// Mitsubishi GX Works2 project: 2023-06-26 #2 생산자동화기능사 14번   PLC: Q03UDV
// 생산자동화기능사

// global labels: Global1
VAR_GLOBAL
  PB1 AT X0 : BOOL;
  PB2 AT X1 : BOOL;
  정지 AT X2 : BOOL;
  공급후진 AT X3 : BOOL;
  공급전진 AT X4 : BOOL;
  가공후진 AT X5 : BOOL;
  가공전진 AT X6 : BOOL;
  송출후진 AT X7 : BOOL;
  송출전진 AT X8 : BOOL;
  배출후진 AT X9 : BOOL;
  배출전진 AT X0A : BOOL;
  매거진 AT X0B : BOOL;
  금속센서 AT X0F : BOOL;
  PB3 AT X10 : BOOL;
  적색 AT Y20 : BOOL;
  황색 AT Y21 : BOOL;
  녹색 AT Y22 : BOOL;
  공급1 AT Y23 : BOOL;
  공급2 AT Y24 : BOOL;
  가공 AT Y25 : BOOL;
  드릴 AT Y26 : BOOL;
  송출 AT Y27 : BOOL;
  배출 AT Y28 : BOOL;
  컨베이어 AT Y29 : BOOL;
END_VAR

PROGRAM 테스트동작
VAR
  PHASE : INT;
END_VAR
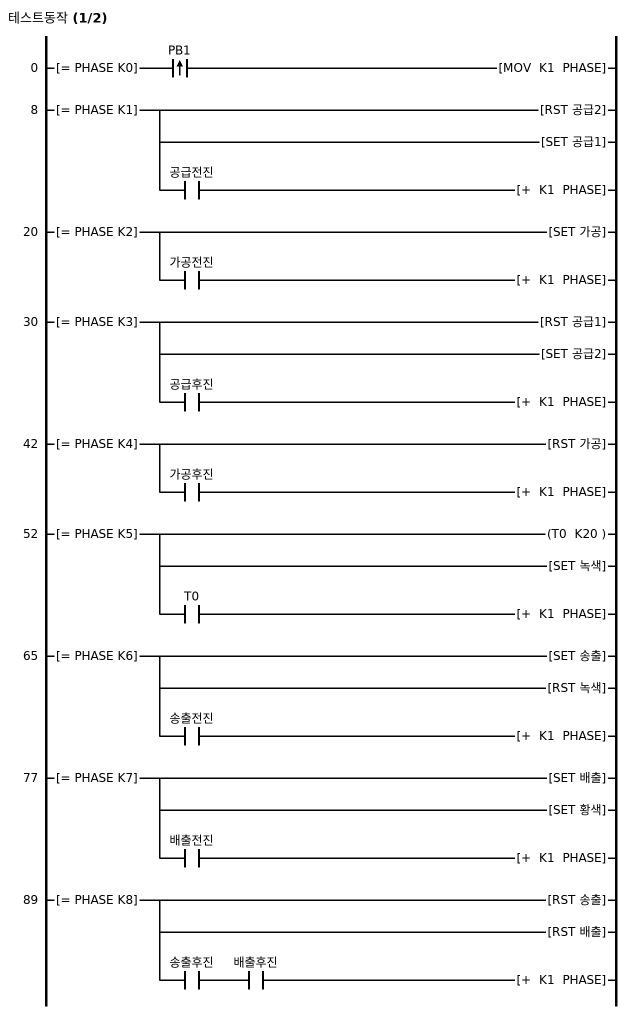
0     LD=     PHASE K0
      ANDP    PB1
      MOV     K1 PHASE
8     LD=     PHASE K1
      RST     공급2
      SET     공급1
      AND     공급전진
      +       K1 PHASE
20    LD=     PHASE K2
      SET     가공
      AND     가공전진
      +       K1 PHASE
30    LD=     PHASE K3
      RST     공급1
      SET     공급2
      AND     공급후진
      +       K1 PHASE
42    LD=     PHASE K4
      RST     가공
      AND     가공후진
      +       K1 PHASE
52    LD=     PHASE K5
      OUT     T0 K20
      SET     녹색
      AND     T0
      +       K1 PHASE
65    LD=     PHASE K6
      SET     송출
      RST     녹색
      AND     송출전진
      +       K1 PHASE
77    LD=     PHASE K7
      SET     배출
      SET     황색
      AND     배출전진
      +       K1 PHASE
89    LD=     PHASE K8
      RST     송출
      RST     배출
      AND     송출후진
      AND     배출후진
      +       K1 PHASE
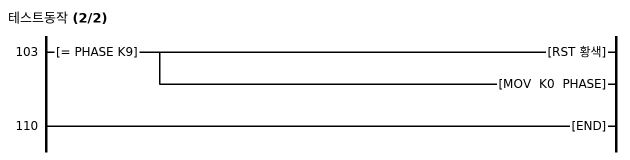
103   LD=     PHASE K9
      RST     황색
      MOV     K0 PHASE
110   END
END_PROGRAM

PROGRAM 단속및연속동작
VAR
  PHASE : INT;
  MODE : INT;
END_VAR
VAR CONSTANT
  단속 : INT;
  연속 : INT := 1;
END_VAR
VAR
  METAL : INT;
END_VAR
VAR CONSTANT
  금속 : INT := 1;
  비금속 : INT := 2;
END_VAR
VAR
  BLINK : ARRAY [0..7] OF BOOL;
  EMG : INT;
END_VAR
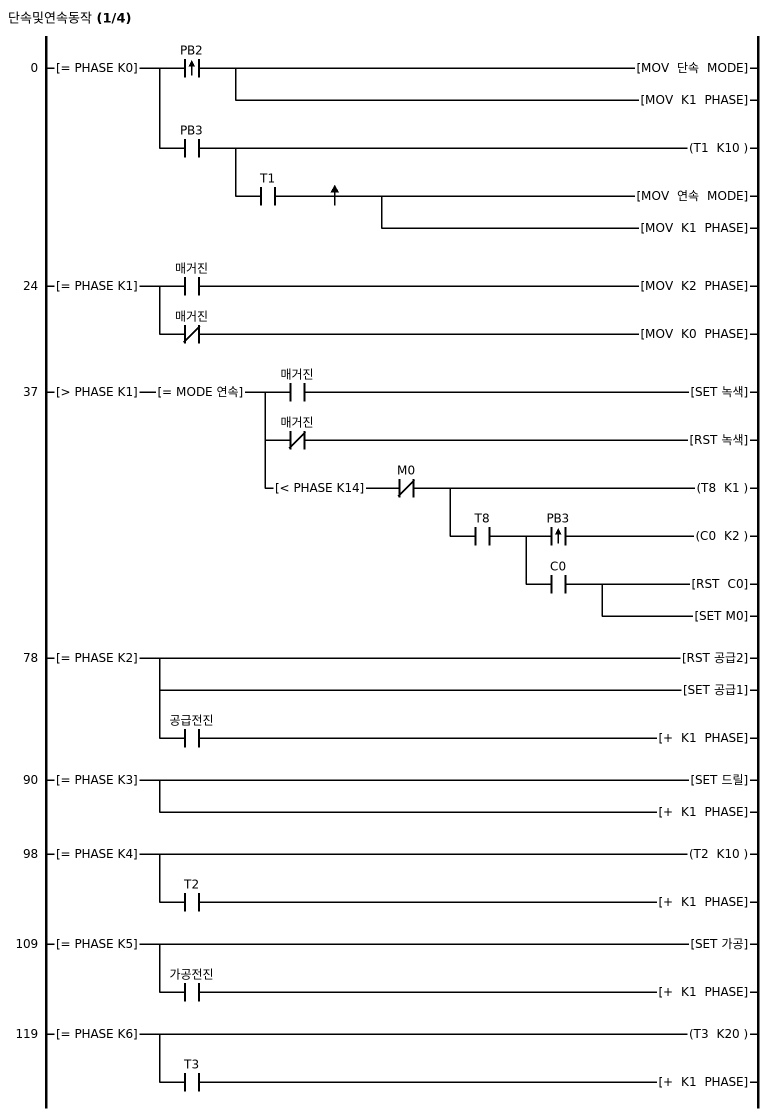
0     LD=     PHASE K0
      MPS
      ANDP    PB2
      MOV     단속 MODE
      MOV     K1 PHASE
      MPP
      AND     PB3
      OUT     T1 K10
      AND     T1
      MEP
      MOV     연속 MODE
      MOV     K1 PHASE
24    LD=     PHASE K1
      MPS
      AND     매거진
      MOV     K2 PHASE
      MPP
      ANI     매거진
      MOV     K0 PHASE
37    LD>     PHASE K1
      AND=    MODE 연속
      MPS
      AND     매거진
      SET     녹색
      MRD
      ANI     매거진
      RST     녹색
      MPP
      AND<    PHASE K14
      ANI     M0
      OUT     T8 K1
      AND     T8
      MPS
      ANDP    PB3
      OUT     C0 K2
      MPP
      AND     C0
      RST     C0
      SET     M0
78    LD=     PHASE K2
      RST     공급2
      SET     공급1
      AND     공급전진
      +       K1 PHASE
90    LD=     PHASE K3
      SET     드릴
      +       K1 PHASE
98    LD=     PHASE K4
      OUT     T2 K10
      AND     T2
      +       K1 PHASE
109   LD=     PHASE K5
      SET     가공
      AND     가공전진
      +       K1 PHASE
119   LD=     PHASE K6
      OUT     T3 K20
      AND     T3
      +       K1 PHASE
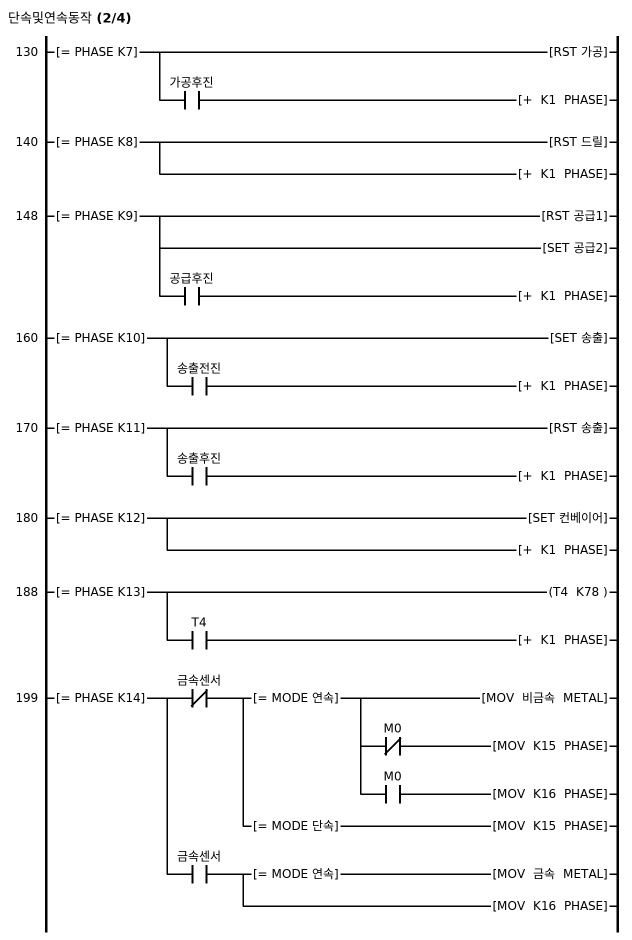
130   LD=     PHASE K7
      RST     가공
      AND     가공후진
      +       K1 PHASE
140   LD=     PHASE K8
      RST     드릴
      +       K1 PHASE
148   LD=     PHASE K9
      RST     공급1
      SET     공급2
      AND     공급후진
      +       K1 PHASE
160   LD=     PHASE K10
      SET     송출
      AND     송출전진
      +       K1 PHASE
170   LD=     PHASE K11
      RST     송출
      AND     송출후진
      +       K1 PHASE
180   LD=     PHASE K12
      SET     컨베이어
      +       K1 PHASE
188   LD=     PHASE K13
      OUT     T4 K78
      AND     T4
      +       K1 PHASE
199   LD=     PHASE K14
      MPS
      ANI     금속센서
      MPS
      AND=    MODE 연속
      MOV     비금속 METAL
      MPS
      ANI     M0
      MOV     K15 PHASE
      MPP
      AND     M0
      MOV     K16 PHASE
      MPP
      AND=    MODE 단속
      MOV     K15 PHASE
      MPP
      AND     금속센서
      MPS
      AND=    MODE 연속
      MOV     금속 METAL
      MPP
      MOV     K16 PHASE
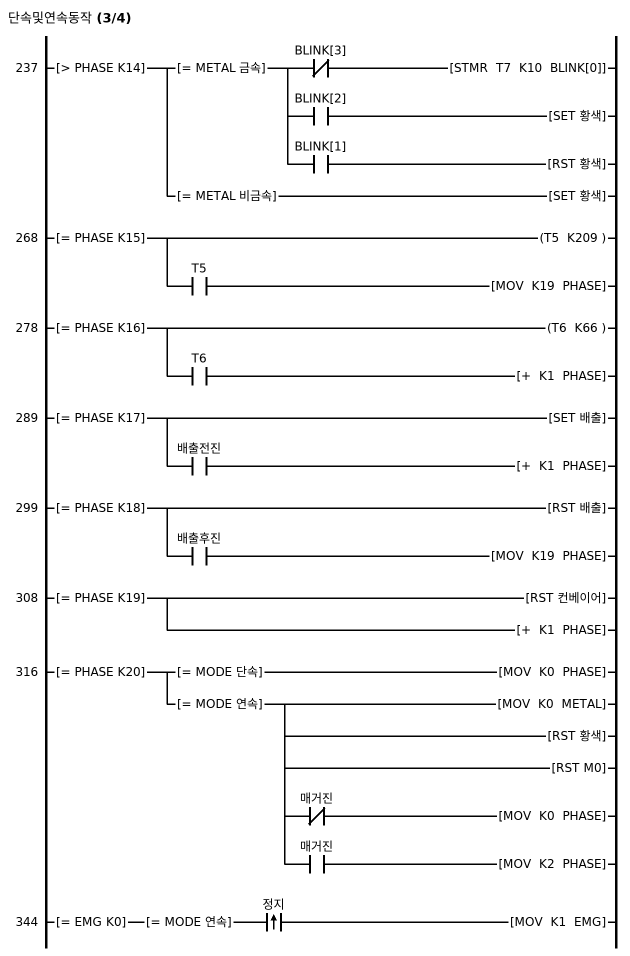
237   LD>     PHASE K14
      MPS
      AND=    METAL 금속
      MPS
      ANI     BLINK[3]
      STMR    T7 K10 BLINK[0]
      MRD
      AND     BLINK[2]
      SET     황색
      MPP
      AND     BLINK[1]
      RST     황색
      MPP
      AND=    METAL 비금속
      SET     황색
268   LD=     PHASE K15
      OUT     T5 K209
      AND     T5
      MOV     K19 PHASE
278   LD=     PHASE K16
      OUT     T6 K66
      AND     T6
      +       K1 PHASE
289   LD=     PHASE K17
      SET     배출
      AND     배출전진
      +       K1 PHASE
299   LD=     PHASE K18
      RST     배출
      AND     배출후진
      MOV     K19 PHASE
308   LD=     PHASE K19
      RST     컨베이어
      +       K1 PHASE
316   LD=     PHASE K20
      MPS
      AND=    MODE 단속
      MOV     K0 PHASE
      MPP
      AND=    MODE 연속
      MOV     K0 METAL
      RST     황색
      RST     M0
      MPS
      ANI     매거진
      MOV     K0 PHASE
      MPP
      AND     매거진
      MOV     K2 PHASE
344   LD=     EMG K0
      AND=    MODE 연속
      ANDP    정지
      MOV     K1 EMG
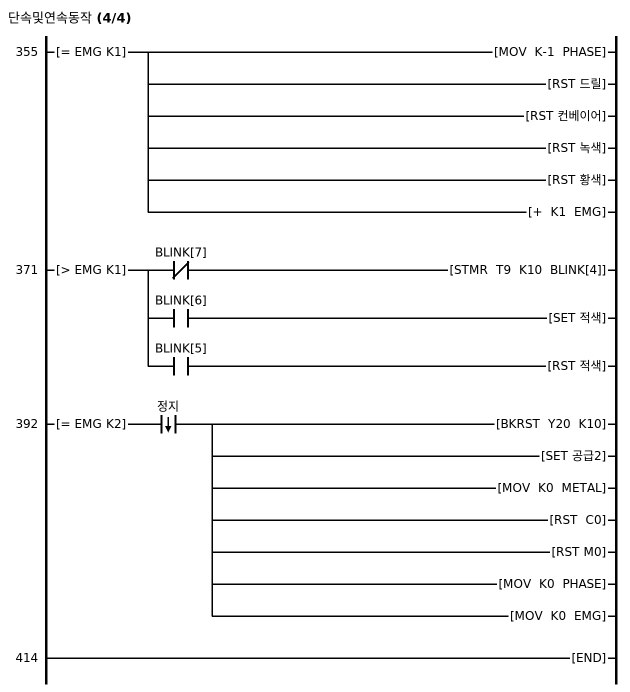
355   LD=     EMG K1
      MOV     K-1 PHASE
      RST     드릴
      RST     컨베이어
      RST     녹색
      RST     황색
      +       K1 EMG
371   LD>     EMG K1
      MPS
      ANI     BLINK[7]
      STMR    T9 K10 BLINK[4]
      MRD
      AND     BLINK[6]
      SET     적색
      MPP
      AND     BLINK[5]
      RST     적색
392   LD=     EMG K2
      ANDF    정지
      BKRST   Y20 K10
      SET     공급2
      MOV     K0 METAL
      RST     C0
      RST     M0
      MOV     K0 PHASE
      MOV     K0 EMG
414   END
END_PROGRAM
